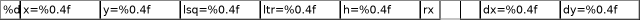
VISUALIZATION _VISU_MarkTriangle_Detail  // 640x20
VAR_IN_OUT
	mInst : ST_MarkDefinition;
END_VAR
    Rectangle (20,0 80x20), "x=%0.4f", text variable: mInst.fPosX
        OnMouseClick: write the text variable via Default
    Rectangle (100,0 80x20), "y=%0.4f", text variable: mInst.fPosY
        OnMouseClick: write the text variable via Default
    RoundedRectangle (460,0 20x20)
        toggle mInst.sState.bSet
    Rectangle (480,0 80x20), "dx=%0.4f", text variable: minst.sState.dx
        OnMouseClick: write the text variable via Default
    Rectangle (560,0 80x20), "dy=%0.4f", text variable: minst.sState.dy
        OnMouseClick: write the text variable via Default
    Rectangle (0,0 20x20), "%d", text variable: mInst.nId, colour toggle: mInst.nId > 0
    RoundedRectangle (420,0 20x20), "rx"
        toggle mInst.bInvertedX
    Rectangle (260,0 80x20), "ltr=%0.4f", text variable: mInst.fTrLength
        OnMouseClick: write the text variable via Default
    Rectangle (340,0 80x20), "h=%0.4f", text variable: mInst.fHeight
        OnMouseClick: write the text variable via Default
    Rectangle (180,0 80x20), "lsq=%0.4f", text variable: mInst.fSqLength
        OnMouseClick: write the text variable via Default
END_VISUALIZATION

(* stored: Version 1.1.0.1, ProductVersion 3.1.4024.11
   Visu _VISU_MarkTriangle_Detail: Id {56b5417a-e213-4767-b24f-f331ad38564b} *)
